PROGRAM MAIN
VAR
END_VAR

END_PROGRAM

(* stored: Version 1.1.0.1
   POU MAIN: Id {5a8e1327-26d3-4e43-8559-97c135f86653} *)
